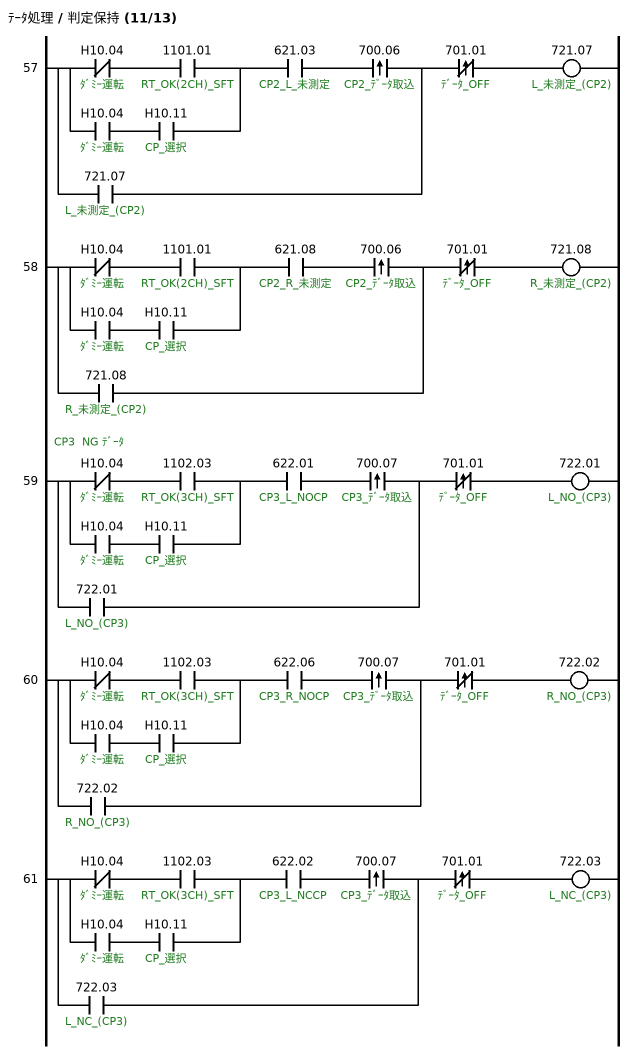
; [picture p144: ﾃｰﾀ処理 / 判定保持, rungs 57-61]
; rung 57
LDNOT H10.04  ; ﾀﾞﾐｰ運転
AND 1101.01  ; RT_OK(2CH)_SFT
LD H10.04  ; ﾀﾞﾐｰ運転
AND H10.11  ; CP_選択
ORLD
AND 621.03  ; CP2_L_未測定
@AND 700.06  ; CP2_ﾃﾞｰﾀ取込
OR 721.07  ; L_未測定_(CP2)
@ANDNOT 701.01  ; ﾃﾞｰﾀ_OFF
OUT 721.07  ; L_未測定_(CP2)
; rung 58
LDNOT H10.04  ; ﾀﾞﾐｰ運転
AND 1101.01  ; RT_OK(2CH)_SFT
LD H10.04  ; ﾀﾞﾐｰ運転
AND H10.11  ; CP_選択
ORLD
AND 621.08  ; CP2_R_未測定
@AND 700.06  ; CP2_ﾃﾞｰﾀ取込
OR 721.08  ; R_未測定_(CP2)
@ANDNOT 701.01  ; ﾃﾞｰﾀ_OFF
OUT 721.08  ; R_未測定_(CP2)
; rung 59: CP3  NG ﾃﾞｰﾀ
LDNOT H10.04  ; ﾀﾞﾐｰ運転
AND 1102.03  ; RT_OK(3CH)_SFT
LD H10.04  ; ﾀﾞﾐｰ運転
AND H10.11  ; CP_選択
ORLD
AND 622.01  ; CP3_L_NOCP
@AND 700.07  ; CP3_ﾃﾞｰﾀ取込
OR 722.01  ; L_NO_(CP3)
@ANDNOT 701.01  ; ﾃﾞｰﾀ_OFF
OUT 722.01  ; L_NO_(CP3)
; rung 60
LDNOT H10.04  ; ﾀﾞﾐｰ運転
AND 1102.03  ; RT_OK(3CH)_SFT
LD H10.04  ; ﾀﾞﾐｰ運転
AND H10.11  ; CP_選択
ORLD
AND 622.06  ; CP3_R_NOCP
@AND 700.07  ; CP3_ﾃﾞｰﾀ取込
OR 722.02  ; R_NO_(CP3)
@ANDNOT 701.01  ; ﾃﾞｰﾀ_OFF
OUT 722.02  ; R_NO_(CP3)
; rung 61
LDNOT H10.04  ; ﾀﾞﾐｰ運転
AND 1102.03  ; RT_OK(3CH)_SFT
LD H10.04  ; ﾀﾞﾐｰ運転
AND H10.11  ; CP_選択
ORLD
AND 622.02  ; CP3_L_NCCP
@AND 700.07  ; CP3_ﾃﾞｰﾀ取込
OR 722.03  ; L_NC_(CP3)
@ANDNOT 701.01  ; ﾃﾞｰﾀ_OFF
OUT 722.03  ; L_NC_(CP3)

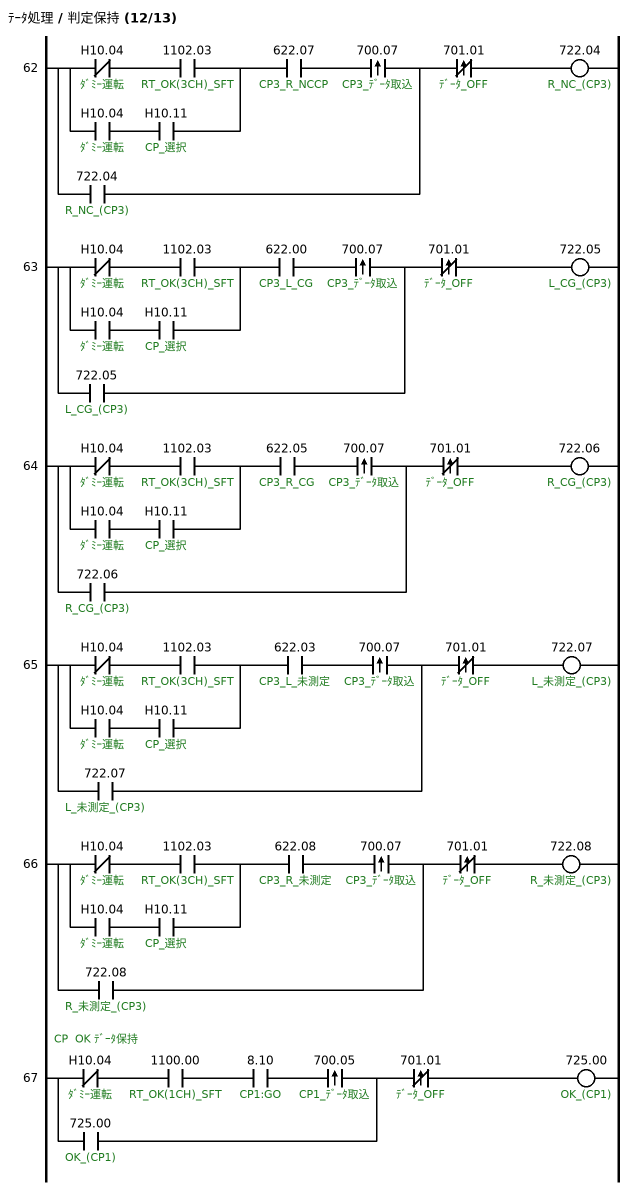
; rung 62
LDNOT H10.04  ; ﾀﾞﾐｰ運転
AND 1102.03  ; RT_OK(3CH)_SFT
LD H10.04  ; ﾀﾞﾐｰ運転
AND H10.11  ; CP_選択
ORLD
AND 622.07  ; CP3_R_NCCP
@AND 700.07  ; CP3_ﾃﾞｰﾀ取込
OR 722.04  ; R_NC_(CP3)
@ANDNOT 701.01  ; ﾃﾞｰﾀ_OFF
OUT 722.04  ; R_NC_(CP3)
; rung 63
LDNOT H10.04  ; ﾀﾞﾐｰ運転
AND 1102.03  ; RT_OK(3CH)_SFT
LD H10.04  ; ﾀﾞﾐｰ運転
AND H10.11  ; CP_選択
ORLD
AND 622.00  ; CP3_L_CG
@AND 700.07  ; CP3_ﾃﾞｰﾀ取込
OR 722.05  ; L_CG_(CP3)
@ANDNOT 701.01  ; ﾃﾞｰﾀ_OFF
OUT 722.05  ; L_CG_(CP3)
; rung 64
LDNOT H10.04  ; ﾀﾞﾐｰ運転
AND 1102.03  ; RT_OK(3CH)_SFT
LD H10.04  ; ﾀﾞﾐｰ運転
AND H10.11  ; CP_選択
ORLD
AND 622.05  ; CP3_R_CG
@AND 700.07  ; CP3_ﾃﾞｰﾀ取込
OR 722.06  ; R_CG_(CP3)
@ANDNOT 701.01  ; ﾃﾞｰﾀ_OFF
OUT 722.06  ; R_CG_(CP3)
; rung 65
LDNOT H10.04  ; ﾀﾞﾐｰ運転
AND 1102.03  ; RT_OK(3CH)_SFT
LD H10.04  ; ﾀﾞﾐｰ運転
AND H10.11  ; CP_選択
ORLD
AND 622.03  ; CP3_L_未測定
@AND 700.07  ; CP3_ﾃﾞｰﾀ取込
OR 722.07  ; L_未測定_(CP3)
@ANDNOT 701.01  ; ﾃﾞｰﾀ_OFF
OUT 722.07  ; L_未測定_(CP3)
; rung 66
LDNOT H10.04  ; ﾀﾞﾐｰ運転
AND 1102.03  ; RT_OK(3CH)_SFT
LD H10.04  ; ﾀﾞﾐｰ運転
AND H10.11  ; CP_選択
ORLD
AND 622.08  ; CP3_R_未測定
@AND 700.07  ; CP3_ﾃﾞｰﾀ取込
OR 722.08  ; R_未測定_(CP3)
@ANDNOT 701.01  ; ﾃﾞｰﾀ_OFF
OUT 722.08  ; R_未測定_(CP3)
; rung 67: CP  OK ﾃﾞｰﾀ保持
LDNOT H10.04  ; ﾀﾞﾐｰ運転
AND 1100.00  ; RT_OK(1CH)_SFT
AND 8.10  ; CP1:GO
@AND 700.05  ; CP1_ﾃﾞｰﾀ取込
OR 725.00  ; OK_(CP1)
@ANDNOT 701.01  ; ﾃﾞｰﾀ_OFF
OUT 725.00  ; OK_(CP1)

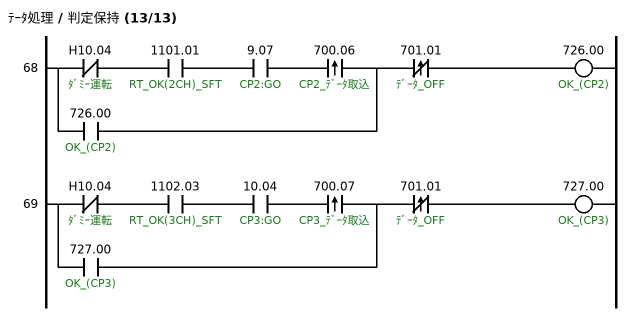
; rung 68
LDNOT H10.04  ; ﾀﾞﾐｰ運転
AND 1101.01  ; RT_OK(2CH)_SFT
AND 9.07  ; CP2:GO
@AND 700.06  ; CP2_ﾃﾞｰﾀ取込
OR 726.00  ; OK_(CP2)
@ANDNOT 701.01  ; ﾃﾞｰﾀ_OFF
OUT 726.00  ; OK_(CP2)
; rung 69
LDNOT H10.04  ; ﾀﾞﾐｰ運転
AND 1102.03  ; RT_OK(3CH)_SFT
AND 10.04  ; CP3:GO
@AND 700.07  ; CP3_ﾃﾞｰﾀ取込
OR 727.00  ; OK_(CP3)
@ANDNOT 701.01  ; ﾃﾞｰﾀ_OFF
OUT 727.00  ; OK_(CP3)

### Section NG_SFT

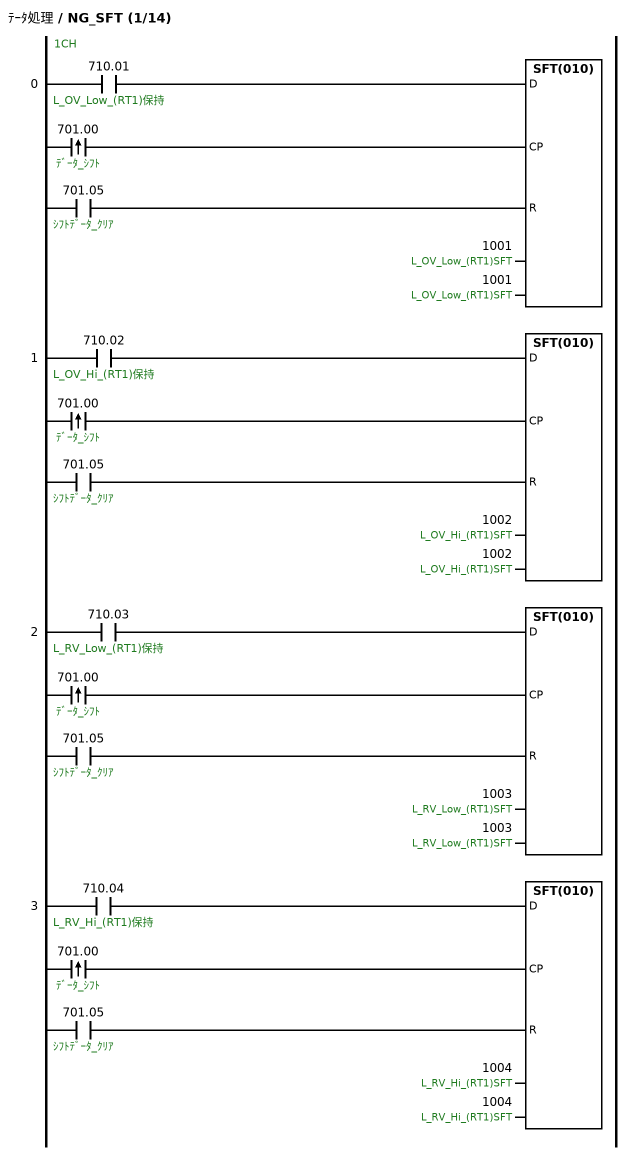
; rung 0: 1CH
LD 710.01  ; L_OV_Low_(RT1)保持
@LD 701.00  ; ﾃﾞｰﾀ_ｼﾌﾄ
LD 701.05  ; ｼﾌﾄﾃﾞｰﾀ_ｸﾘｱ
SFT(010) 1001 1001  ; L_OV_Low_(RT1)SFT
; rung 1
LD 710.02  ; L_OV_Hi_(RT1)保持
@LD 701.00  ; ﾃﾞｰﾀ_ｼﾌﾄ
LD 701.05  ; ｼﾌﾄﾃﾞｰﾀ_ｸﾘｱ
SFT(010) 1002 1002  ; L_OV_Hi_(RT1)SFT
; rung 2
LD 710.03  ; L_RV_Low_(RT1)保持
@LD 701.00  ; ﾃﾞｰﾀ_ｼﾌﾄ
LD 701.05  ; ｼﾌﾄﾃﾞｰﾀ_ｸﾘｱ
SFT(010) 1003 1003  ; L_RV_Low_(RT1)SFT
; rung 3
LD 710.04  ; L_RV_Hi_(RT1)保持
@LD 701.00  ; ﾃﾞｰﾀ_ｼﾌﾄ
LD 701.05  ; ｼﾌﾄﾃﾞｰﾀ_ｸﾘｱ
SFT(010) 1004 1004  ; L_RV_Hi_(RT1)SFT

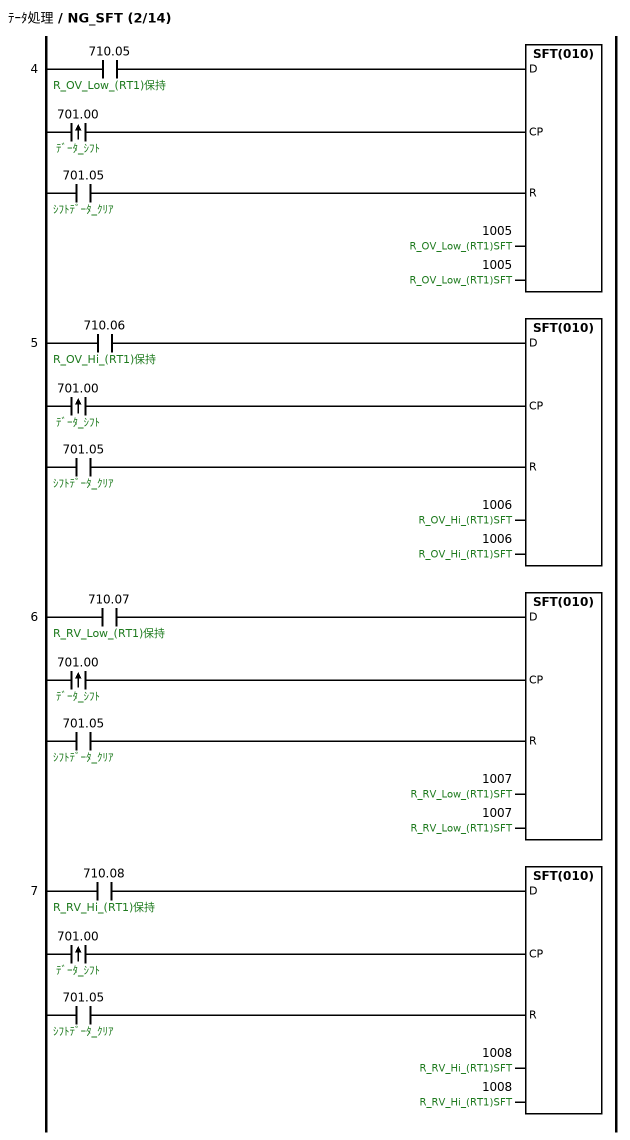
; rung 4
LD 710.05  ; R_OV_Low_(RT1)保持
@LD 701.00  ; ﾃﾞｰﾀ_ｼﾌﾄ
LD 701.05  ; ｼﾌﾄﾃﾞｰﾀ_ｸﾘｱ
SFT(010) 1005 1005  ; R_OV_Low_(RT1)SFT
; rung 5
LD 710.06  ; R_OV_Hi_(RT1)保持
@LD 701.00  ; ﾃﾞｰﾀ_ｼﾌﾄ
LD 701.05  ; ｼﾌﾄﾃﾞｰﾀ_ｸﾘｱ
SFT(010) 1006 1006  ; R_OV_Hi_(RT1)SFT
; rung 6
LD 710.07  ; R_RV_Low_(RT1)保持
@LD 701.00  ; ﾃﾞｰﾀ_ｼﾌﾄ
LD 701.05  ; ｼﾌﾄﾃﾞｰﾀ_ｸﾘｱ
SFT(010) 1007 1007  ; R_RV_Low_(RT1)SFT
; rung 7
LD 710.08  ; R_RV_Hi_(RT1)保持
@LD 701.00  ; ﾃﾞｰﾀ_ｼﾌﾄ
LD 701.05  ; ｼﾌﾄﾃﾞｰﾀ_ｸﾘｱ
SFT(010) 1008 1008  ; R_RV_Hi_(RT1)SFT

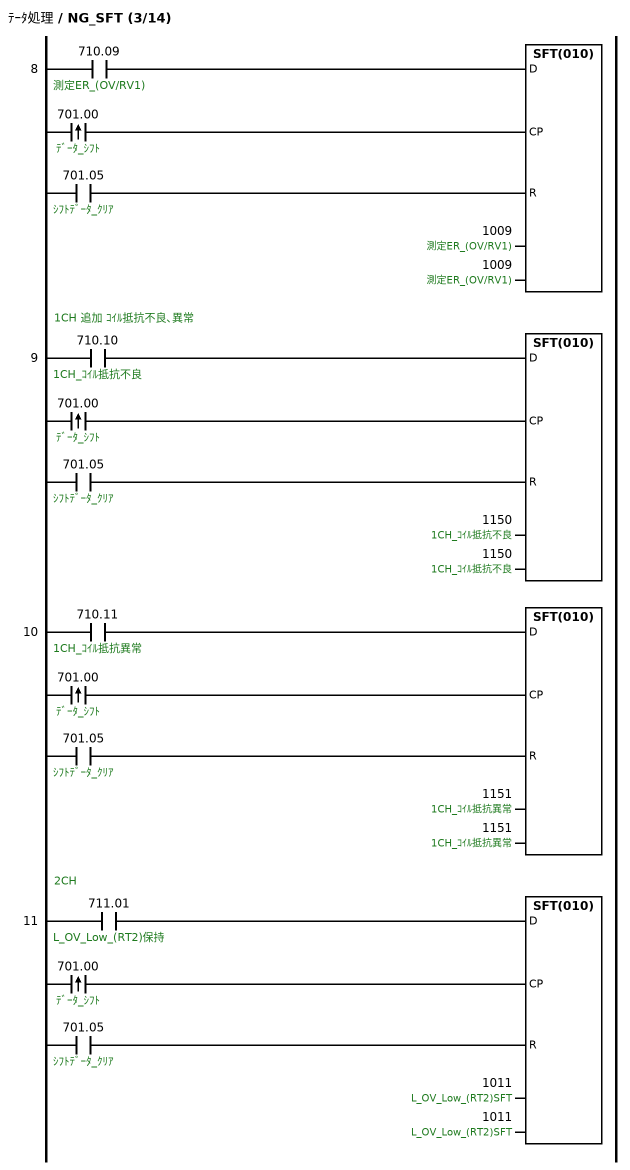
; rung 8
LD 710.09  ; 測定ER_(OV/RV1)
@LD 701.00  ; ﾃﾞｰﾀ_ｼﾌﾄ
LD 701.05  ; ｼﾌﾄﾃﾞｰﾀ_ｸﾘｱ
SFT(010) 1009 1009  ; 測定ER_(OV/RV1)
; rung 9: 1CH 追加 ｺｲﾙ抵抗不良､異常
LD 710.10  ; 1CH_ｺｲﾙ抵抗不良
@LD 701.00  ; ﾃﾞｰﾀ_ｼﾌﾄ
LD 701.05  ; ｼﾌﾄﾃﾞｰﾀ_ｸﾘｱ
SFT(010) 1150 1150  ; 1CH_ｺｲﾙ抵抗不良
; rung 10
LD 710.11  ; 1CH_ｺｲﾙ抵抗異常
@LD 701.00  ; ﾃﾞｰﾀ_ｼﾌﾄ
LD 701.05  ; ｼﾌﾄﾃﾞｰﾀ_ｸﾘｱ
SFT(010) 1151 1151  ; 1CH_ｺｲﾙ抵抗異常
; rung 11: 2CH
LD 711.01  ; L_OV_Low_(RT2)保持
@LD 701.00  ; ﾃﾞｰﾀ_ｼﾌﾄ
LD 701.05  ; ｼﾌﾄﾃﾞｰﾀ_ｸﾘｱ
SFT(010) 1011 1011  ; L_OV_Low_(RT2)SFT

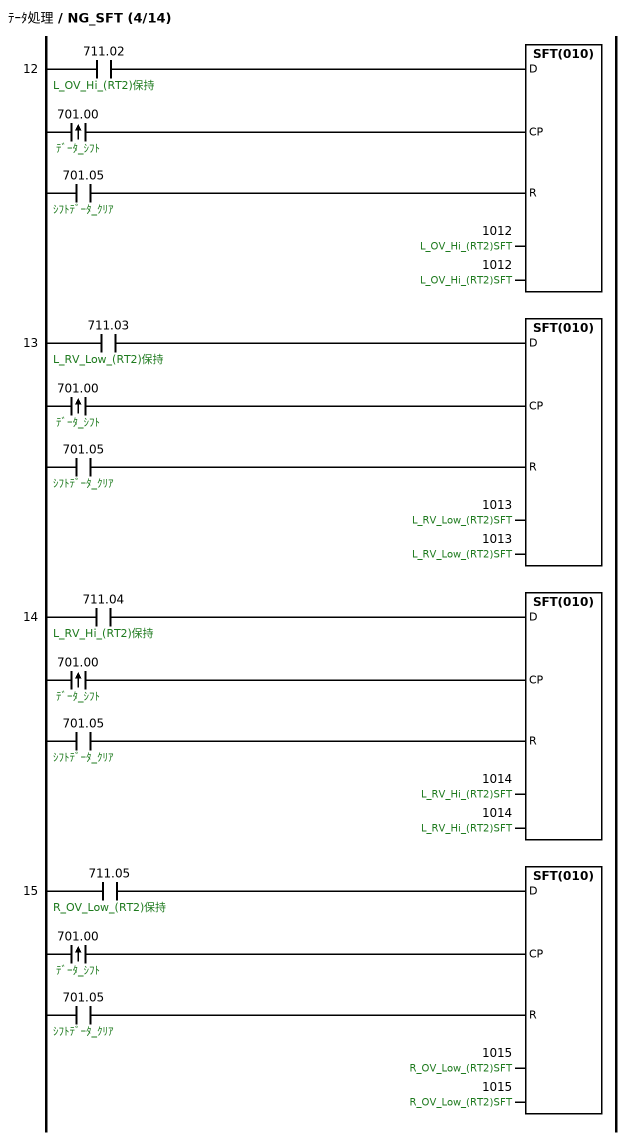
; rung 12
LD 711.02  ; L_OV_Hi_(RT2)保持
@LD 701.00  ; ﾃﾞｰﾀ_ｼﾌﾄ
LD 701.05  ; ｼﾌﾄﾃﾞｰﾀ_ｸﾘｱ
SFT(010) 1012 1012  ; L_OV_Hi_(RT2)SFT
; rung 13
LD 711.03  ; L_RV_Low_(RT2)保持
@LD 701.00  ; ﾃﾞｰﾀ_ｼﾌﾄ
LD 701.05  ; ｼﾌﾄﾃﾞｰﾀ_ｸﾘｱ
SFT(010) 1013 1013  ; L_RV_Low_(RT2)SFT
; rung 14
LD 711.04  ; L_RV_Hi_(RT2)保持
@LD 701.00  ; ﾃﾞｰﾀ_ｼﾌﾄ
LD 701.05  ; ｼﾌﾄﾃﾞｰﾀ_ｸﾘｱ
SFT(010) 1014 1014  ; L_RV_Hi_(RT2)SFT
; rung 15
LD 711.05  ; R_OV_Low_(RT2)保持
@LD 701.00  ; ﾃﾞｰﾀ_ｼﾌﾄ
LD 701.05  ; ｼﾌﾄﾃﾞｰﾀ_ｸﾘｱ
SFT(010) 1015 1015  ; R_OV_Low_(RT2)SFT

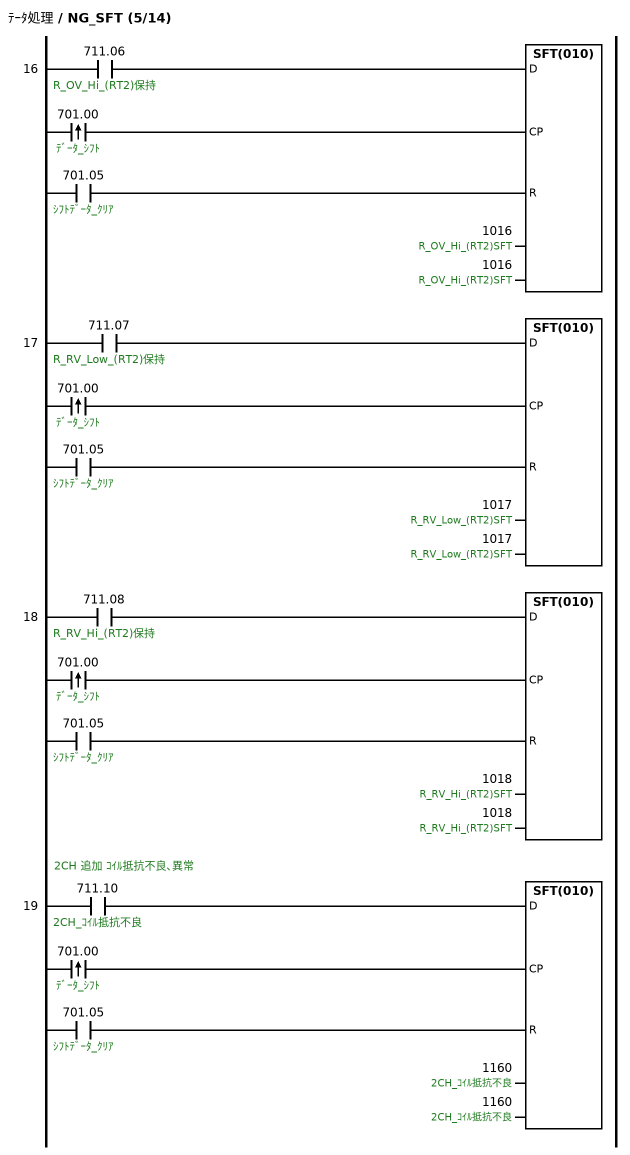
; rung 16
LD 711.06  ; R_OV_Hi_(RT2)保持
@LD 701.00  ; ﾃﾞｰﾀ_ｼﾌﾄ
LD 701.05  ; ｼﾌﾄﾃﾞｰﾀ_ｸﾘｱ
SFT(010) 1016 1016  ; R_OV_Hi_(RT2)SFT
; rung 17
LD 711.07  ; R_RV_Low_(RT2)保持
@LD 701.00  ; ﾃﾞｰﾀ_ｼﾌﾄ
LD 701.05  ; ｼﾌﾄﾃﾞｰﾀ_ｸﾘｱ
SFT(010) 1017 1017  ; R_RV_Low_(RT2)SFT
; rung 18
LD 711.08  ; R_RV_Hi_(RT2)保持
@LD 701.00  ; ﾃﾞｰﾀ_ｼﾌﾄ
LD 701.05  ; ｼﾌﾄﾃﾞｰﾀ_ｸﾘｱ
SFT(010) 1018 1018  ; R_RV_Hi_(RT2)SFT
; rung 19: 2CH 追加 ｺｲﾙ抵抗不良､異常
LD 711.10  ; 2CH_ｺｲﾙ抵抗不良
@LD 701.00  ; ﾃﾞｰﾀ_ｼﾌﾄ
LD 701.05  ; ｼﾌﾄﾃﾞｰﾀ_ｸﾘｱ
SFT(010) 1160 1160  ; 2CH_ｺｲﾙ抵抗不良

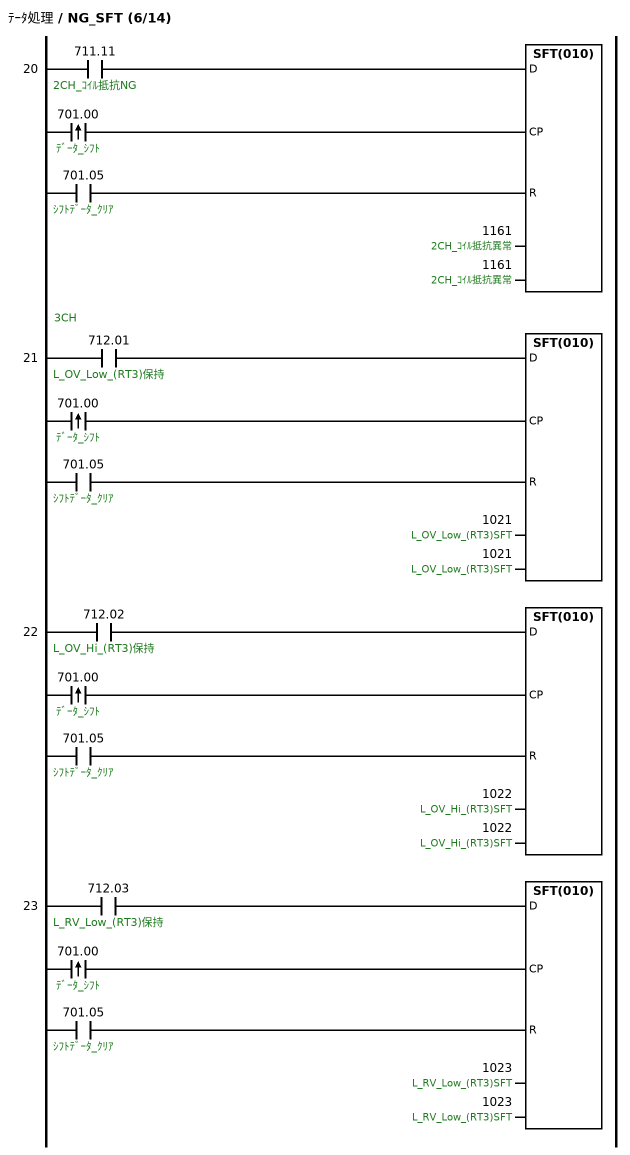
; rung 20
LD 711.11  ; 2CH_ｺｲﾙ抵抗NG
@LD 701.00  ; ﾃﾞｰﾀ_ｼﾌﾄ
LD 701.05  ; ｼﾌﾄﾃﾞｰﾀ_ｸﾘｱ
SFT(010) 1161 1161  ; 2CH_ｺｲﾙ抵抗異常
; rung 21: 3CH
LD 712.01  ; L_OV_Low_(RT3)保持
@LD 701.00  ; ﾃﾞｰﾀ_ｼﾌﾄ
LD 701.05  ; ｼﾌﾄﾃﾞｰﾀ_ｸﾘｱ
SFT(010) 1021 1021  ; L_OV_Low_(RT3)SFT
; rung 22
LD 712.02  ; L_OV_Hi_(RT3)保持
@LD 701.00  ; ﾃﾞｰﾀ_ｼﾌﾄ
LD 701.05  ; ｼﾌﾄﾃﾞｰﾀ_ｸﾘｱ
SFT(010) 1022 1022  ; L_OV_Hi_(RT3)SFT
; rung 23
LD 712.03  ; L_RV_Low_(RT3)保持
@LD 701.00  ; ﾃﾞｰﾀ_ｼﾌﾄ
LD 701.05  ; ｼﾌﾄﾃﾞｰﾀ_ｸﾘｱ
SFT(010) 1023 1023  ; L_RV_Low_(RT3)SFT

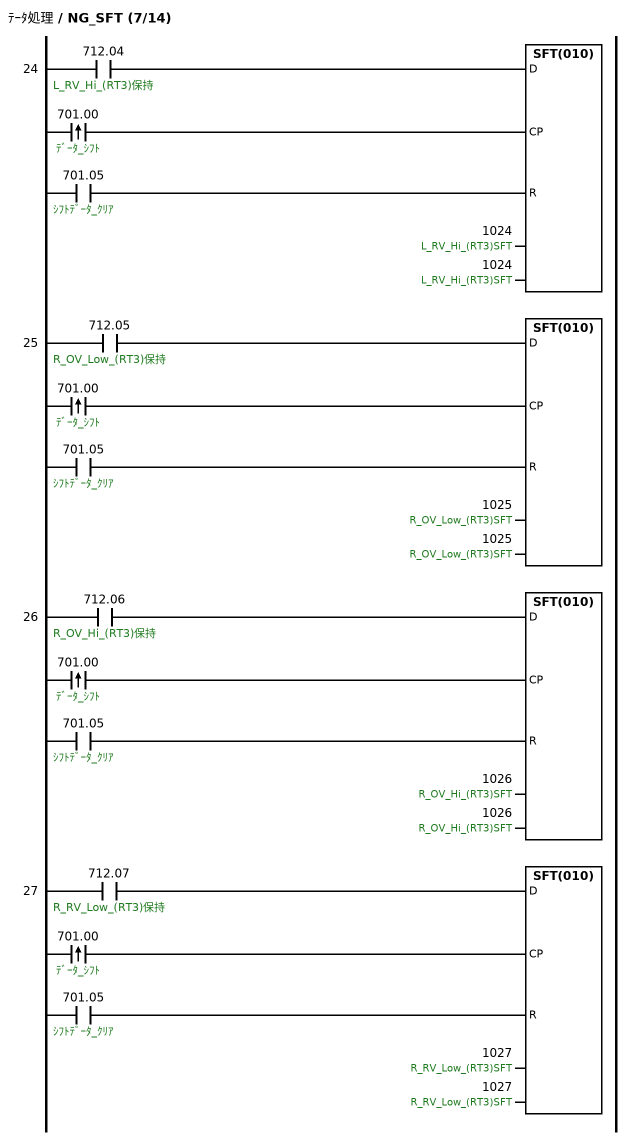
; rung 24
LD 712.04  ; L_RV_Hi_(RT3)保持
@LD 701.00  ; ﾃﾞｰﾀ_ｼﾌﾄ
LD 701.05  ; ｼﾌﾄﾃﾞｰﾀ_ｸﾘｱ
SFT(010) 1024 1024  ; L_RV_Hi_(RT3)SFT
; rung 25
LD 712.05  ; R_OV_Low_(RT3)保持
@LD 701.00  ; ﾃﾞｰﾀ_ｼﾌﾄ
LD 701.05  ; ｼﾌﾄﾃﾞｰﾀ_ｸﾘｱ
SFT(010) 1025 1025  ; R_OV_Low_(RT3)SFT
; rung 26
LD 712.06  ; R_OV_Hi_(RT3)保持
@LD 701.00  ; ﾃﾞｰﾀ_ｼﾌﾄ
LD 701.05  ; ｼﾌﾄﾃﾞｰﾀ_ｸﾘｱ
SFT(010) 1026 1026  ; R_OV_Hi_(RT3)SFT
; rung 27
LD 712.07  ; R_RV_Low_(RT3)保持
@LD 701.00  ; ﾃﾞｰﾀ_ｼﾌﾄ
LD 701.05  ; ｼﾌﾄﾃﾞｰﾀ_ｸﾘｱ
SFT(010) 1027 1027  ; R_RV_Low_(RT3)SFT

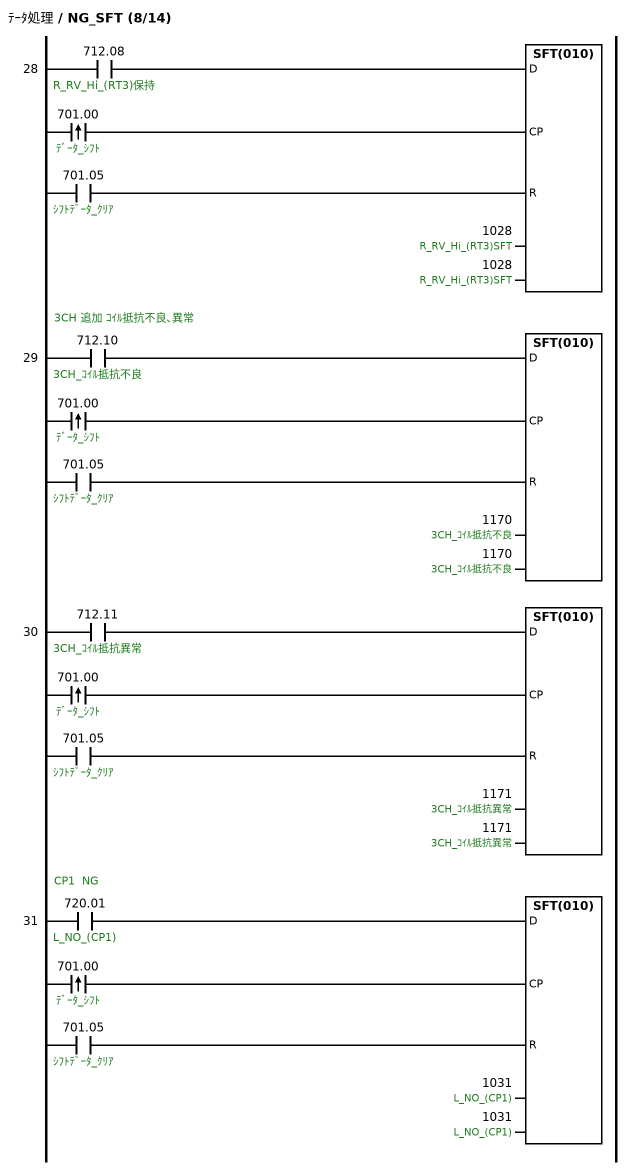
; rung 28
LD 712.08  ; R_RV_Hi_(RT3)保持
@LD 701.00  ; ﾃﾞｰﾀ_ｼﾌﾄ
LD 701.05  ; ｼﾌﾄﾃﾞｰﾀ_ｸﾘｱ
SFT(010) 1028 1028  ; R_RV_Hi_(RT3)SFT
; rung 29: 3CH 追加 ｺｲﾙ抵抗不良､異常
LD 712.10  ; 3CH_ｺｲﾙ抵抗不良
@LD 701.00  ; ﾃﾞｰﾀ_ｼﾌﾄ
LD 701.05  ; ｼﾌﾄﾃﾞｰﾀ_ｸﾘｱ
SFT(010) 1170 1170  ; 3CH_ｺｲﾙ抵抗不良
; rung 30
LD 712.11  ; 3CH_ｺｲﾙ抵抗異常
@LD 701.00  ; ﾃﾞｰﾀ_ｼﾌﾄ
LD 701.05  ; ｼﾌﾄﾃﾞｰﾀ_ｸﾘｱ
SFT(010) 1171 1171  ; 3CH_ｺｲﾙ抵抗異常
; rung 31: CP1  NG
LD 720.01  ; L_NO_(CP1)
@LD 701.00  ; ﾃﾞｰﾀ_ｼﾌﾄ
LD 701.05  ; ｼﾌﾄﾃﾞｰﾀ_ｸﾘｱ
SFT(010) 1031 1031  ; L_NO_(CP1)

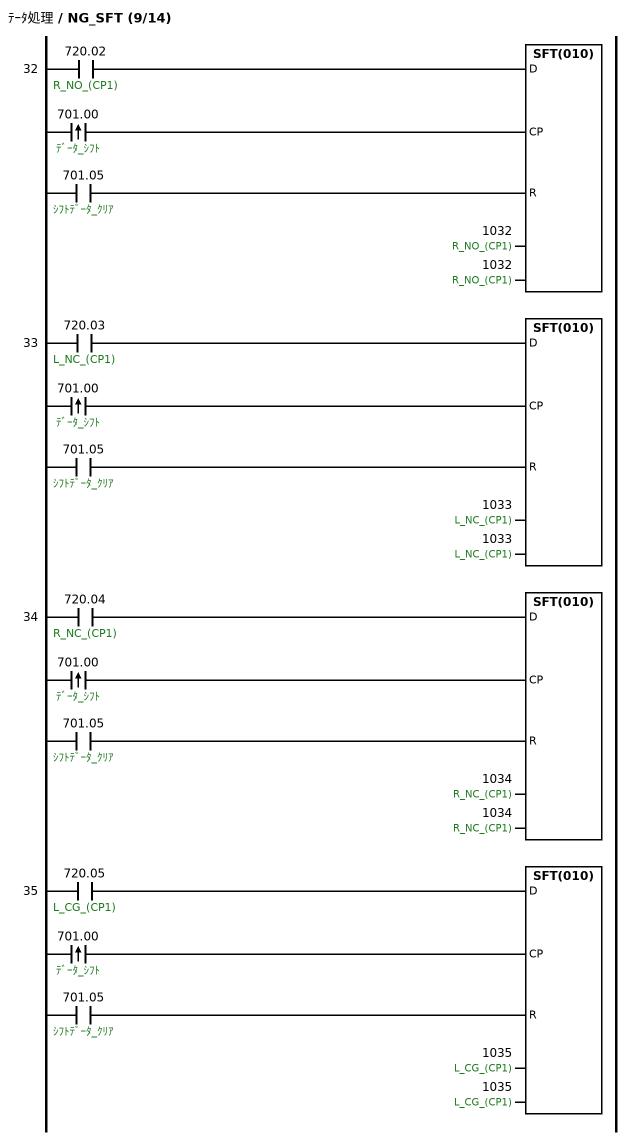
; rung 32
LD 720.02  ; R_NO_(CP1)
@LD 701.00  ; ﾃﾞｰﾀ_ｼﾌﾄ
LD 701.05  ; ｼﾌﾄﾃﾞｰﾀ_ｸﾘｱ
SFT(010) 1032 1032  ; R_NO_(CP1)
; rung 33
LD 720.03  ; L_NC_(CP1)
@LD 701.00  ; ﾃﾞｰﾀ_ｼﾌﾄ
LD 701.05  ; ｼﾌﾄﾃﾞｰﾀ_ｸﾘｱ
SFT(010) 1033 1033  ; L_NC_(CP1)
; rung 34
LD 720.04  ; R_NC_(CP1)
@LD 701.00  ; ﾃﾞｰﾀ_ｼﾌﾄ
LD 701.05  ; ｼﾌﾄﾃﾞｰﾀ_ｸﾘｱ
SFT(010) 1034 1034  ; R_NC_(CP1)
; rung 35
LD 720.05  ; L_CG_(CP1)
@LD 701.00  ; ﾃﾞｰﾀ_ｼﾌﾄ
LD 701.05  ; ｼﾌﾄﾃﾞｰﾀ_ｸﾘｱ
SFT(010) 1035 1035  ; L_CG_(CP1)

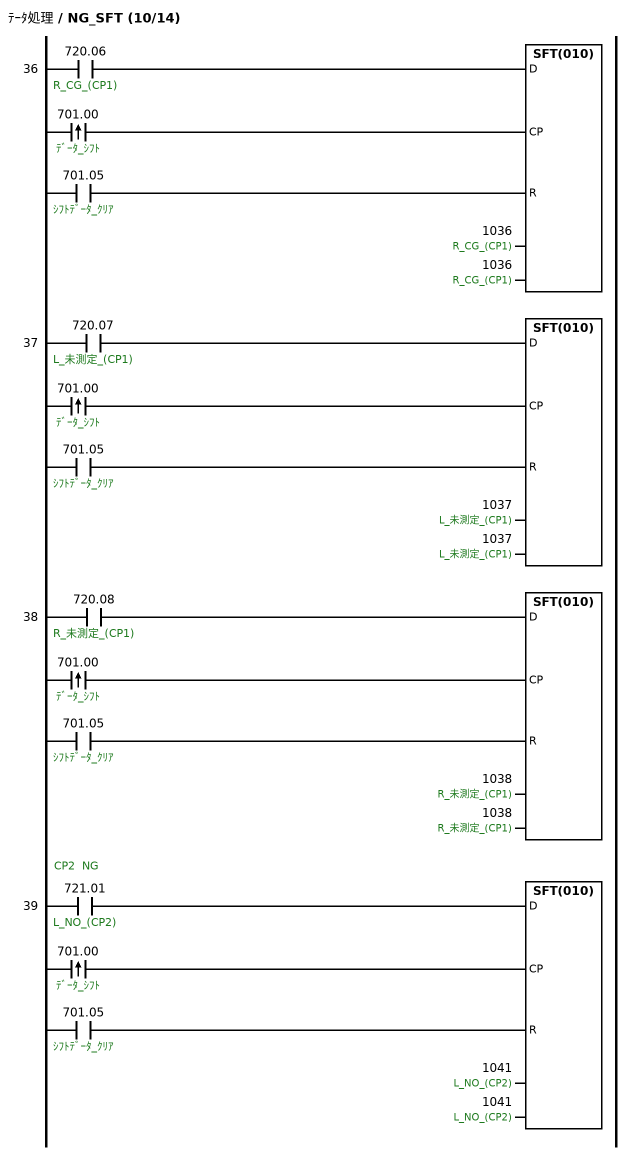
; rung 36
LD 720.06  ; R_CG_(CP1)
@LD 701.00  ; ﾃﾞｰﾀ_ｼﾌﾄ
LD 701.05  ; ｼﾌﾄﾃﾞｰﾀ_ｸﾘｱ
SFT(010) 1036 1036  ; R_CG_(CP1)
; rung 37
LD 720.07  ; L_未測定_(CP1)
@LD 701.00  ; ﾃﾞｰﾀ_ｼﾌﾄ
LD 701.05  ; ｼﾌﾄﾃﾞｰﾀ_ｸﾘｱ
SFT(010) 1037 1037  ; L_未測定_(CP1)
; rung 38
LD 720.08  ; R_未測定_(CP1)
@LD 701.00  ; ﾃﾞｰﾀ_ｼﾌﾄ
LD 701.05  ; ｼﾌﾄﾃﾞｰﾀ_ｸﾘｱ
SFT(010) 1038 1038  ; R_未測定_(CP1)
; rung 39: CP2  NG
LD 721.01  ; L_NO_(CP2)
@LD 701.00  ; ﾃﾞｰﾀ_ｼﾌﾄ
LD 701.05  ; ｼﾌﾄﾃﾞｰﾀ_ｸﾘｱ
SFT(010) 1041 1041  ; L_NO_(CP2)

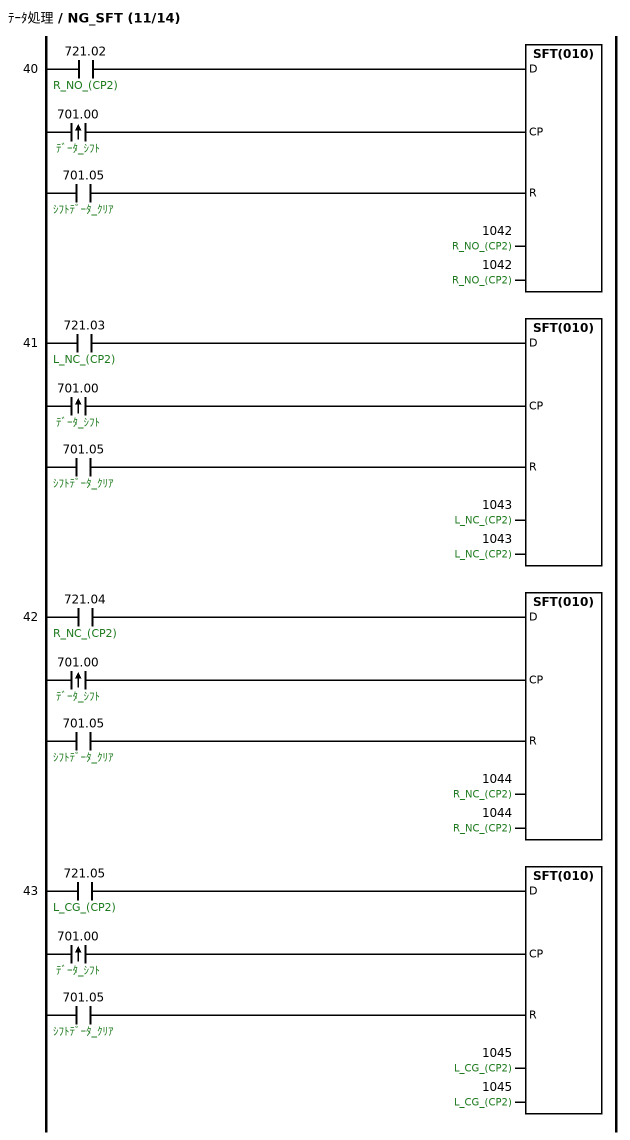
; rung 40
LD 721.02  ; R_NO_(CP2)
@LD 701.00  ; ﾃﾞｰﾀ_ｼﾌﾄ
LD 701.05  ; ｼﾌﾄﾃﾞｰﾀ_ｸﾘｱ
SFT(010) 1042 1042  ; R_NO_(CP2)
; rung 41
LD 721.03  ; L_NC_(CP2)
@LD 701.00  ; ﾃﾞｰﾀ_ｼﾌﾄ
LD 701.05  ; ｼﾌﾄﾃﾞｰﾀ_ｸﾘｱ
SFT(010) 1043 1043  ; L_NC_(CP2)
; rung 42
LD 721.04  ; R_NC_(CP2)
@LD 701.00  ; ﾃﾞｰﾀ_ｼﾌﾄ
LD 701.05  ; ｼﾌﾄﾃﾞｰﾀ_ｸﾘｱ
SFT(010) 1044 1044  ; R_NC_(CP2)
; rung 43
LD 721.05  ; L_CG_(CP2)
@LD 701.00  ; ﾃﾞｰﾀ_ｼﾌﾄ
LD 701.05  ; ｼﾌﾄﾃﾞｰﾀ_ｸﾘｱ
SFT(010) 1045 1045  ; L_CG_(CP2)

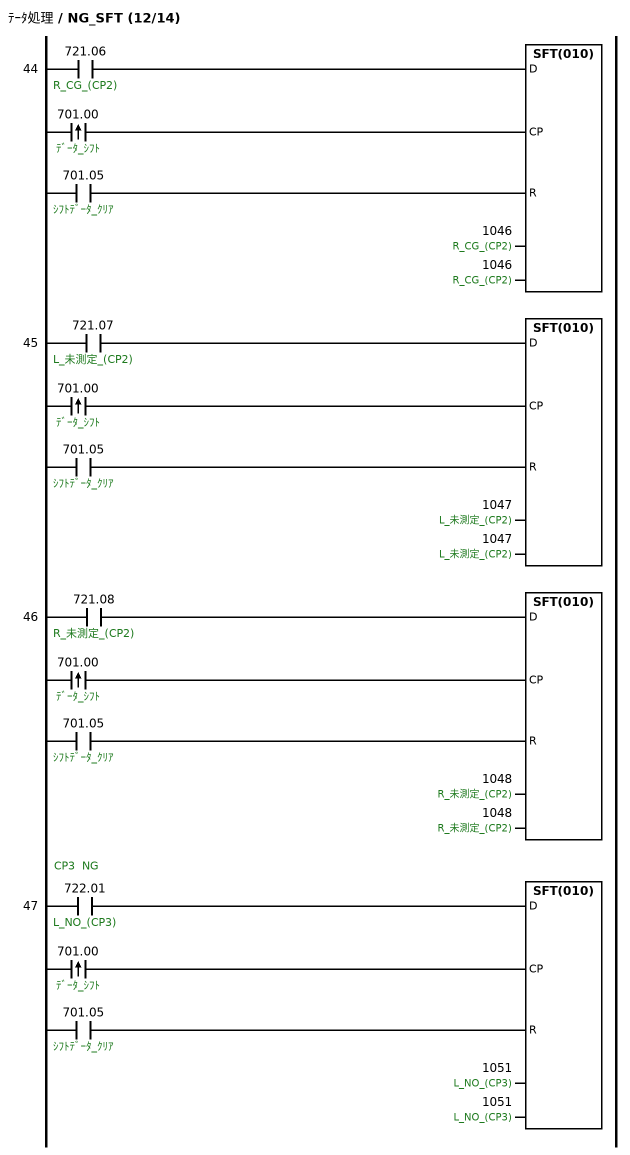
; rung 44
LD 721.06  ; R_CG_(CP2)
@LD 701.00  ; ﾃﾞｰﾀ_ｼﾌﾄ
LD 701.05  ; ｼﾌﾄﾃﾞｰﾀ_ｸﾘｱ
SFT(010) 1046 1046  ; R_CG_(CP2)
; rung 45
LD 721.07  ; L_未測定_(CP2)
@LD 701.00  ; ﾃﾞｰﾀ_ｼﾌﾄ
LD 701.05  ; ｼﾌﾄﾃﾞｰﾀ_ｸﾘｱ
SFT(010) 1047 1047  ; L_未測定_(CP2)
; rung 46
LD 721.08  ; R_未測定_(CP2)
@LD 701.00  ; ﾃﾞｰﾀ_ｼﾌﾄ
LD 701.05  ; ｼﾌﾄﾃﾞｰﾀ_ｸﾘｱ
SFT(010) 1048 1048  ; R_未測定_(CP2)
; rung 47: CP3  NG
LD 722.01  ; L_NO_(CP3)
@LD 701.00  ; ﾃﾞｰﾀ_ｼﾌﾄ
LD 701.05  ; ｼﾌﾄﾃﾞｰﾀ_ｸﾘｱ
SFT(010) 1051 1051  ; L_NO_(CP3)

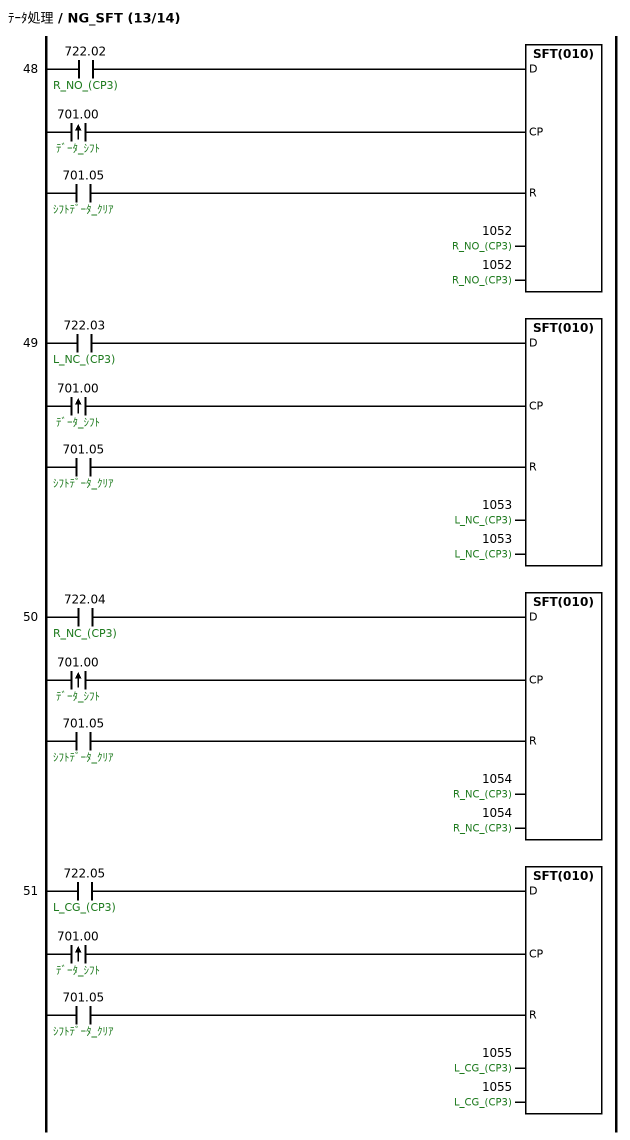
; rung 48
LD 722.02  ; R_NO_(CP3)
@LD 701.00  ; ﾃﾞｰﾀ_ｼﾌﾄ
LD 701.05  ; ｼﾌﾄﾃﾞｰﾀ_ｸﾘｱ
SFT(010) 1052 1052  ; R_NO_(CP3)
; rung 49
LD 722.03  ; L_NC_(CP3)
@LD 701.00  ; ﾃﾞｰﾀ_ｼﾌﾄ
LD 701.05  ; ｼﾌﾄﾃﾞｰﾀ_ｸﾘｱ
SFT(010) 1053 1053  ; L_NC_(CP3)
; rung 50
LD 722.04  ; R_NC_(CP3)
@LD 701.00  ; ﾃﾞｰﾀ_ｼﾌﾄ
LD 701.05  ; ｼﾌﾄﾃﾞｰﾀ_ｸﾘｱ
SFT(010) 1054 1054  ; R_NC_(CP3)
; rung 51
LD 722.05  ; L_CG_(CP3)
@LD 701.00  ; ﾃﾞｰﾀ_ｼﾌﾄ
LD 701.05  ; ｼﾌﾄﾃﾞｰﾀ_ｸﾘｱ
SFT(010) 1055 1055  ; L_CG_(CP3)

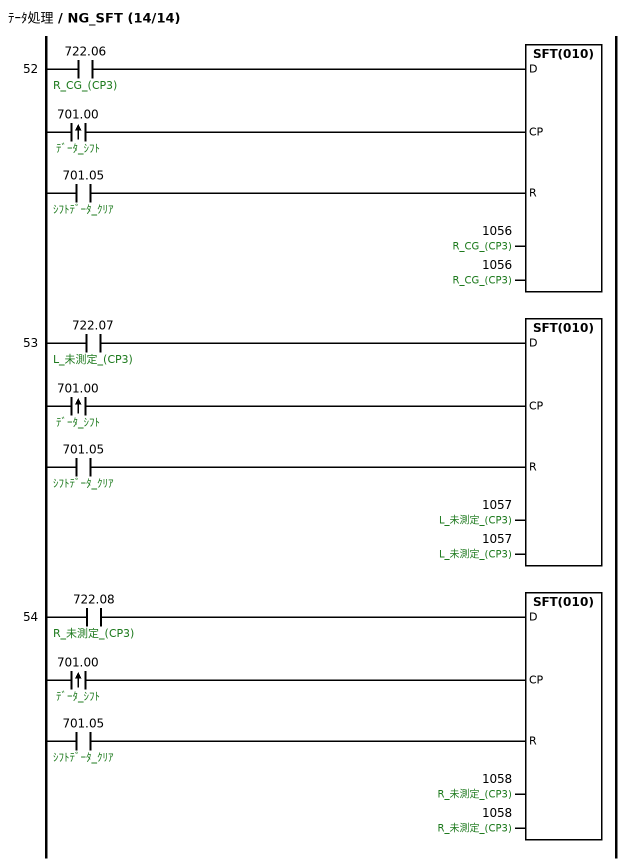
; rung 52
LD 722.06  ; R_CG_(CP3)
@LD 701.00  ; ﾃﾞｰﾀ_ｼﾌﾄ
LD 701.05  ; ｼﾌﾄﾃﾞｰﾀ_ｸﾘｱ
SFT(010) 1056 1056  ; R_CG_(CP3)
; rung 53
LD 722.07  ; L_未測定_(CP3)
@LD 701.00  ; ﾃﾞｰﾀ_ｼﾌﾄ
LD 701.05  ; ｼﾌﾄﾃﾞｰﾀ_ｸﾘｱ
SFT(010) 1057 1057  ; L_未測定_(CP3)
; rung 54
LD 722.08  ; R_未測定_(CP3)
@LD 701.00  ; ﾃﾞｰﾀ_ｼﾌﾄ
LD 701.05  ; ｼﾌﾄﾃﾞｰﾀ_ｸﾘｱ
SFT(010) 1058 1058  ; R_未測定_(CP3)

### Section OK_SFT

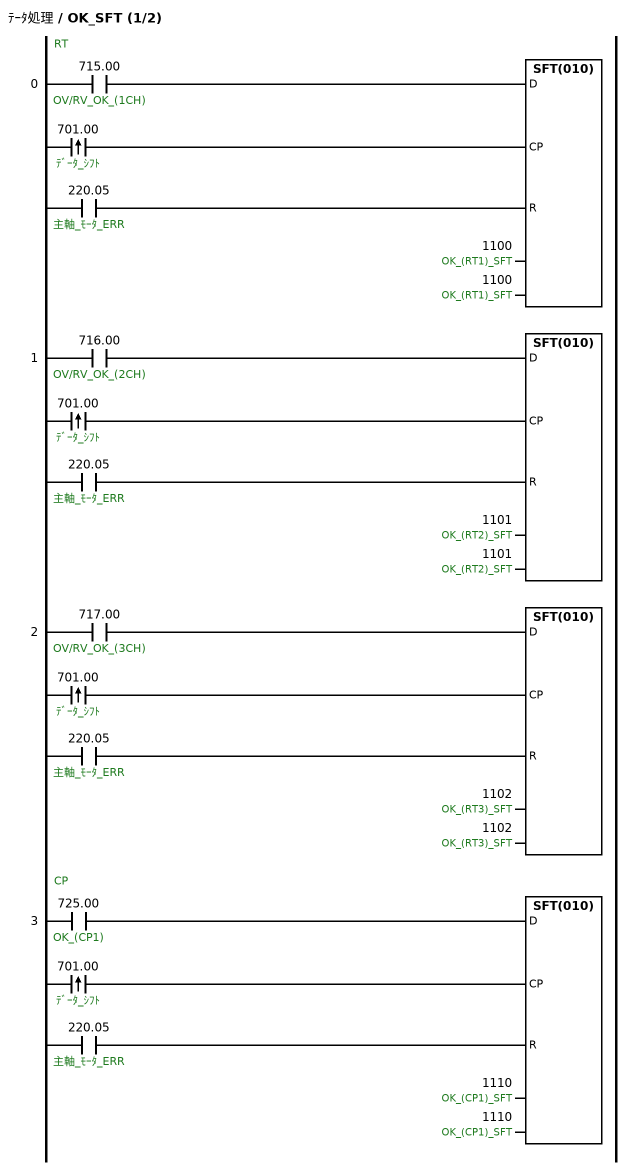
; rung 0: RT
LD 715.00  ; OV/RV_OK_(1CH)
@LD 701.00  ; ﾃﾞｰﾀ_ｼﾌﾄ
LD 220.05  ; 主軸_ﾓｰﾀ_ERR
SFT(010) 1100 1100  ; OK_(RT1)_SFT
; rung 1
LD 716.00  ; OV/RV_OK_(2CH)
@LD 701.00  ; ﾃﾞｰﾀ_ｼﾌﾄ
LD 220.05  ; 主軸_ﾓｰﾀ_ERR
SFT(010) 1101 1101  ; OK_(RT2)_SFT
; rung 2
LD 717.00  ; OV/RV_OK_(3CH)
@LD 701.00  ; ﾃﾞｰﾀ_ｼﾌﾄ
LD 220.05  ; 主軸_ﾓｰﾀ_ERR
SFT(010) 1102 1102  ; OK_(RT3)_SFT
; rung 3: CP
LD 725.00  ; OK_(CP1)
@LD 701.00  ; ﾃﾞｰﾀ_ｼﾌﾄ
LD 220.05  ; 主軸_ﾓｰﾀ_ERR
SFT(010) 1110 1110  ; OK_(CP1)_SFT

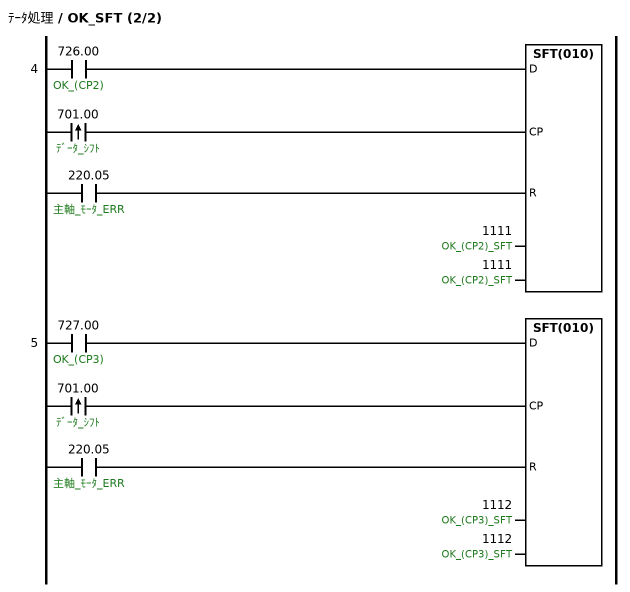
; rung 4
LD 726.00  ; OK_(CP2)
@LD 701.00  ; ﾃﾞｰﾀ_ｼﾌﾄ
LD 220.05  ; 主軸_ﾓｰﾀ_ERR
SFT(010) 1111 1111  ; OK_(CP2)_SFT
; rung 5
LD 727.00  ; OK_(CP3)
@LD 701.00  ; ﾃﾞｰﾀ_ｼﾌﾄ
LD 220.05  ; 主軸_ﾓｰﾀ_ERR
SFT(010) 1112 1112  ; OK_(CP3)_SFT

### Section ﾃﾞｰﾀ処理

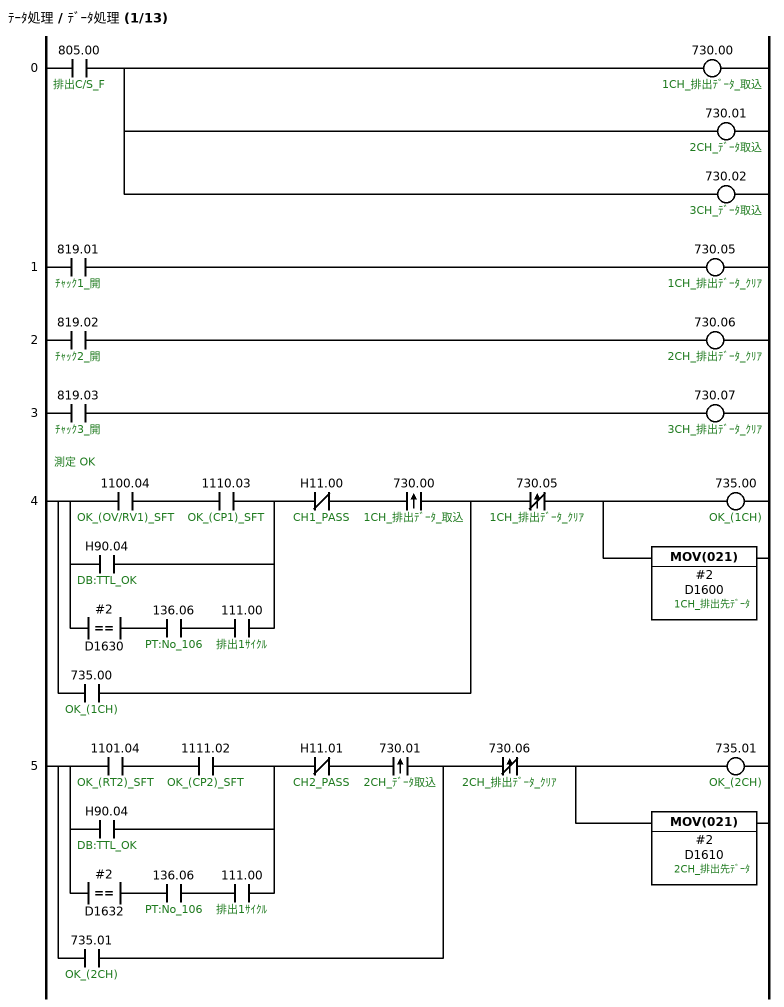
; rung 0
LD 805.00  ; 排出C/S_F
OUT 730.00  ; 1CH_排出ﾃﾞｰﾀ_取込
OUT 730.01  ; 2CH_ﾃﾞｰﾀ取込
OUT 730.02  ; 3CH_ﾃﾞｰﾀ取込
; rung 1
LD 819.01  ; ﾁｬｯｸ1_開
OUT 730.05  ; 1CH_排出ﾃﾞｰﾀ_ｸﾘｱ
; rung 2
LD 819.02  ; ﾁｬｯｸ2_開
OUT 730.06  ; 2CH_排出ﾃﾞｰﾀ_ｸﾘｱ
; rung 3
LD 819.03  ; ﾁｬｯｸ3_開
OUT 730.07  ; 3CH_排出ﾃﾞｰﾀ_ｸﾘｱ
; rung 4: 測定 OK
LD 1100.04  ; OK_(OV/RV1)_SFT
AND 1110.03  ; OK_(CP1)_SFT
OR H90.04  ; DB:TTL_OK
LD=(300) #2 D1630
AND 136.06  ; PT:No_106
AND 111.00  ; 排出1ｻｲｸﾙ
ORLD
ANDNOT H11.00  ; CH1_PASS
@AND 730.00  ; 1CH_排出ﾃﾞｰﾀ_取込
OR 735.00  ; OK_(1CH)
@ANDNOT 730.05  ; 1CH_排出ﾃﾞｰﾀ_ｸﾘｱ
OUT 735.00  ; OK_(1CH)
MOV(021) #2 D1600  ; 1CH_排出先ﾃﾞｰﾀ
; rung 5
LD 1101.04  ; OK_(RT2)_SFT
AND 1111.02  ; OK_(CP2)_SFT
OR H90.04  ; DB:TTL_OK
LD=(300) #2 D1632
AND 136.06  ; PT:No_106
AND 111.00  ; 排出1ｻｲｸﾙ
ORLD
ANDNOT H11.01  ; CH2_PASS
@AND 730.01  ; 2CH_ﾃﾞｰﾀ取込
OR 735.01  ; OK_(2CH)
@ANDNOT 730.06  ; 2CH_排出ﾃﾞｰﾀ_ｸﾘｱ
OUT 735.01  ; OK_(2CH)
MOV(021) #2 D1610  ; 2CH_排出先ﾃﾞｰﾀ

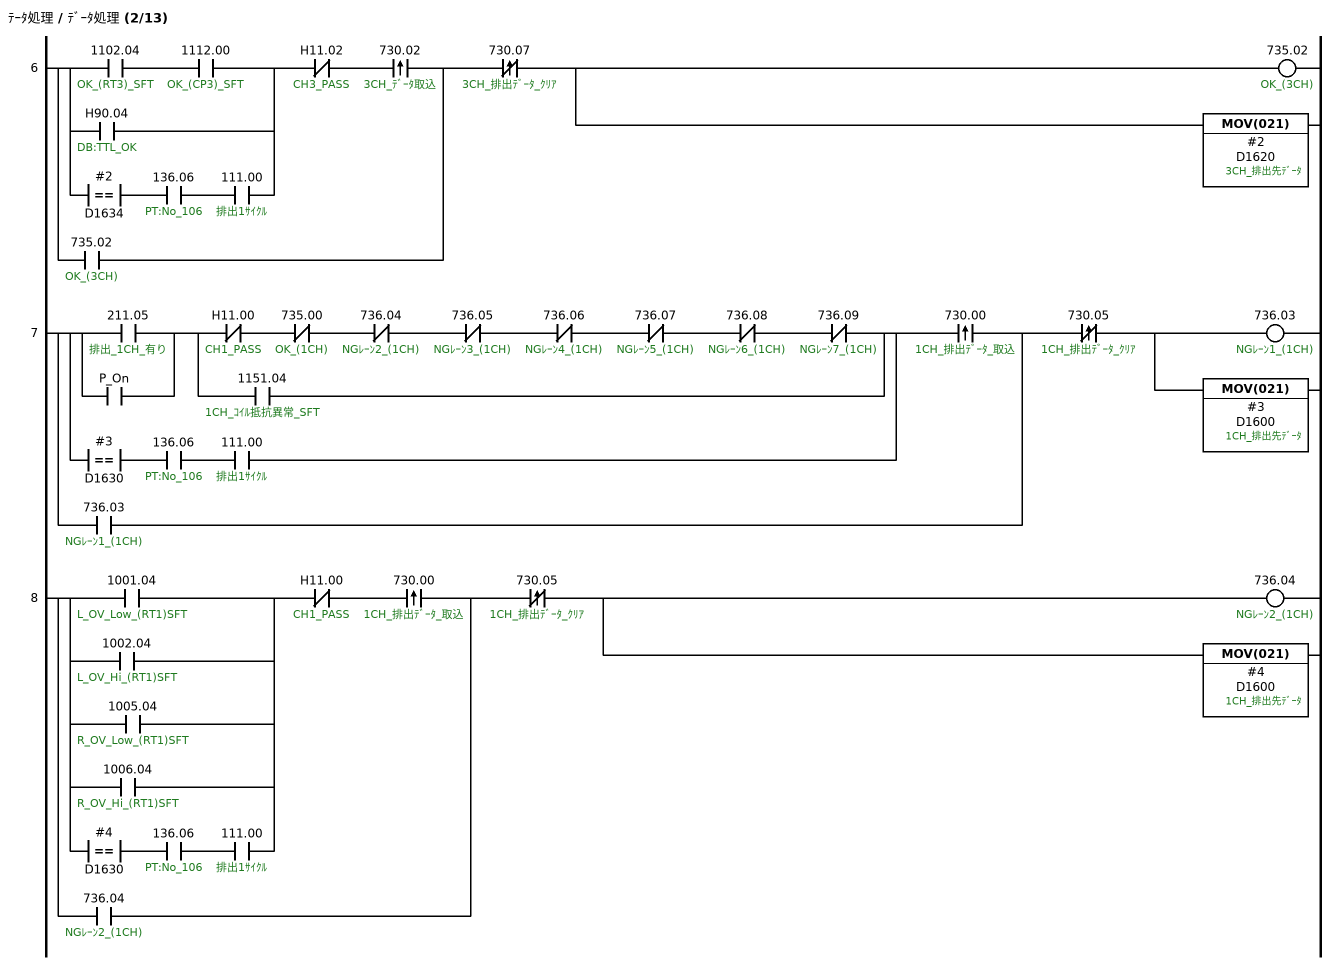
; rung 6
LD 1102.04  ; OK_(RT3)_SFT
AND 1112.00  ; OK_(CP3)_SFT
OR H90.04  ; DB:TTL_OK
LD=(300) #2 D1634
AND 136.06  ; PT:No_106
AND 111.00  ; 排出1ｻｲｸﾙ
ORLD
ANDNOT H11.02  ; CH3_PASS
@AND 730.02  ; 3CH_ﾃﾞｰﾀ取込
OR 735.02  ; OK_(3CH)
@ANDNOT 730.07  ; 3CH_排出ﾃﾞｰﾀ_ｸﾘｱ
OUT 735.02  ; OK_(3CH)
MOV(021) #2 D1620  ; 3CH_排出先ﾃﾞｰﾀ
; rung 7
LD 211.05  ; 排出_1CH_有り
OR P_On
LDNOT H11.00  ; CH1_PASS
ANDNOT 735.00  ; OK_(1CH)
ANDNOT 736.04  ; NGﾚｰﾝ2_(1CH)
ANDNOT 736.05  ; NGﾚｰﾝ3_(1CH)
ANDNOT 736.06  ; NGﾚｰﾝ4_(1CH)
ANDNOT 736.07  ; NGﾚｰﾝ5_(1CH)
ANDNOT 736.08  ; NGﾚｰﾝ6_(1CH)
ANDNOT 736.09  ; NGﾚｰﾝ7_(1CH)
OR 1151.04  ; 1CH_ｺｲﾙ抵抗異常_SFT
ANDLD
LD=(300) #3 D1630
AND 136.06  ; PT:No_106
AND 111.00  ; 排出1ｻｲｸﾙ
ORLD
@AND 730.00  ; 1CH_排出ﾃﾞｰﾀ_取込
OR 736.03  ; NGﾚｰﾝ1_(1CH)
@ANDNOT 730.05  ; 1CH_排出ﾃﾞｰﾀ_ｸﾘｱ
OUT 736.03  ; NGﾚｰﾝ1_(1CH)
MOV(021) #3 D1600  ; 1CH_排出先ﾃﾞｰﾀ
; rung 8
LD 1001.04  ; L_OV_Low_(RT1)SFT
OR 1002.04  ; L_OV_Hi_(RT1)SFT
OR 1005.04  ; R_OV_Low_(RT1)SFT
OR 1006.04  ; R_OV_Hi_(RT1)SFT
LD=(300) #4 D1630
AND 136.06  ; PT:No_106
AND 111.00  ; 排出1ｻｲｸﾙ
ORLD
ANDNOT H11.00  ; CH1_PASS
@AND 730.00  ; 1CH_排出ﾃﾞｰﾀ_取込
OR 736.04  ; NGﾚｰﾝ2_(1CH)
@ANDNOT 730.05  ; 1CH_排出ﾃﾞｰﾀ_ｸﾘｱ
OUT 736.04  ; NGﾚｰﾝ2_(1CH)
MOV(021) #4 D1600  ; 1CH_排出先ﾃﾞｰﾀ

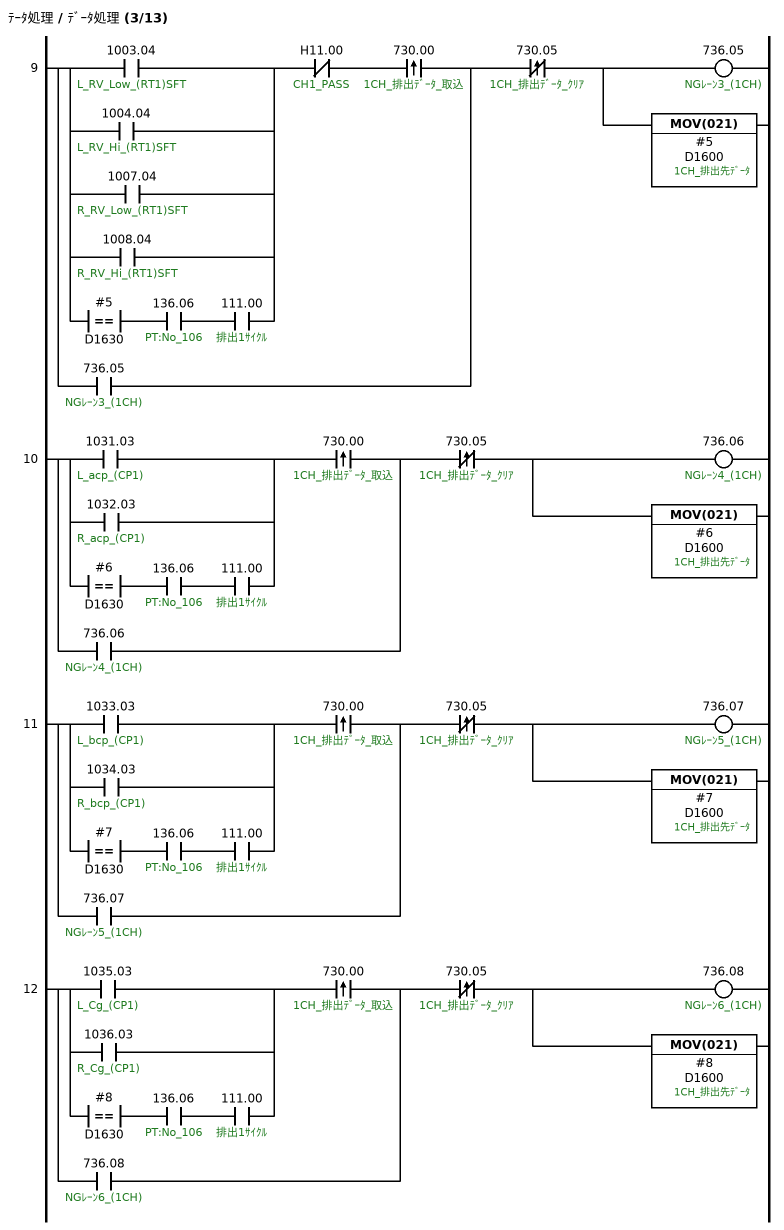
; rung 9
LD 1003.04  ; L_RV_Low_(RT1)SFT
OR 1004.04  ; L_RV_Hi_(RT1)SFT
OR 1007.04  ; R_RV_Low_(RT1)SFT
OR 1008.04  ; R_RV_Hi_(RT1)SFT
LD=(300) #5 D1630
AND 136.06  ; PT:No_106
AND 111.00  ; 排出1ｻｲｸﾙ
ORLD
ANDNOT H11.00  ; CH1_PASS
@AND 730.00  ; 1CH_排出ﾃﾞｰﾀ_取込
OR 736.05  ; NGﾚｰﾝ3_(1CH)
@ANDNOT 730.05  ; 1CH_排出ﾃﾞｰﾀ_ｸﾘｱ
OUT 736.05  ; NGﾚｰﾝ3_(1CH)
MOV(021) #5 D1600  ; 1CH_排出先ﾃﾞｰﾀ
; rung 10
LD 1031.03  ; L_acp_(CP1)
OR 1032.03  ; R_acp_(CP1)
LD=(300) #6 D1630
AND 136.06  ; PT:No_106
AND 111.00  ; 排出1ｻｲｸﾙ
ORLD
@AND 730.00  ; 1CH_排出ﾃﾞｰﾀ_取込
OR 736.06  ; NGﾚｰﾝ4_(1CH)
@ANDNOT 730.05  ; 1CH_排出ﾃﾞｰﾀ_ｸﾘｱ
OUT 736.06  ; NGﾚｰﾝ4_(1CH)
MOV(021) #6 D1600  ; 1CH_排出先ﾃﾞｰﾀ
; rung 11
LD 1033.03  ; L_bcp_(CP1)
OR 1034.03  ; R_bcp_(CP1)
LD=(300) #7 D1630
AND 136.06  ; PT:No_106
AND 111.00  ; 排出1ｻｲｸﾙ
ORLD
@AND 730.00  ; 1CH_排出ﾃﾞｰﾀ_取込
OR 736.07  ; NGﾚｰﾝ5_(1CH)
@ANDNOT 730.05  ; 1CH_排出ﾃﾞｰﾀ_ｸﾘｱ
OUT 736.07  ; NGﾚｰﾝ5_(1CH)
MOV(021) #7 D1600  ; 1CH_排出先ﾃﾞｰﾀ
; rung 12
LD 1035.03  ; L_Cg_(CP1)
OR 1036.03  ; R_Cg_(CP1)
LD=(300) #8 D1630
AND 136.06  ; PT:No_106
AND 111.00  ; 排出1ｻｲｸﾙ
ORLD
@AND 730.00  ; 1CH_排出ﾃﾞｰﾀ_取込
OR 736.08  ; NGﾚｰﾝ6_(1CH)
@ANDNOT 730.05  ; 1CH_排出ﾃﾞｰﾀ_ｸﾘｱ
OUT 736.08  ; NGﾚｰﾝ6_(1CH)
MOV(021) #8 D1600  ; 1CH_排出先ﾃﾞｰﾀ

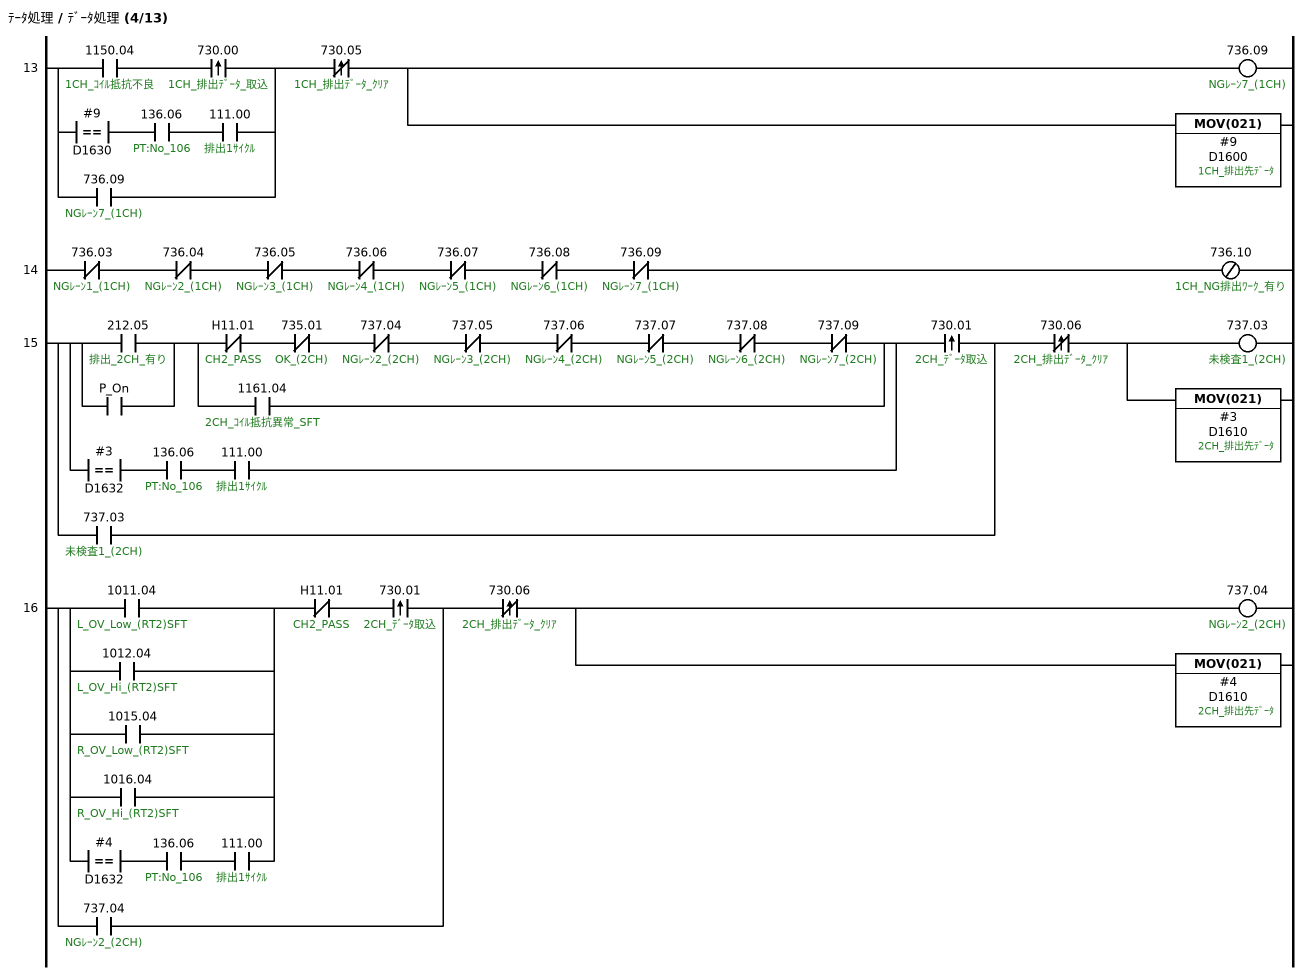
; rung 13
LD 1150.04  ; 1CH_ｺｲﾙ抵抗不良
@AND 730.00  ; 1CH_排出ﾃﾞｰﾀ_取込
LD=(300) #9 D1630
AND 136.06  ; PT:No_106
AND 111.00  ; 排出1ｻｲｸﾙ
ORLD
OR 736.09  ; NGﾚｰﾝ7_(1CH)
@ANDNOT 730.05  ; 1CH_排出ﾃﾞｰﾀ_ｸﾘｱ
OUT 736.09  ; NGﾚｰﾝ7_(1CH)
MOV(021) #9 D1600  ; 1CH_排出先ﾃﾞｰﾀ
; rung 14
LDNOT 736.03  ; NGﾚｰﾝ1_(1CH)
ANDNOT 736.04  ; NGﾚｰﾝ2_(1CH)
ANDNOT 736.05  ; NGﾚｰﾝ3_(1CH)
ANDNOT 736.06  ; NGﾚｰﾝ4_(1CH)
ANDNOT 736.07  ; NGﾚｰﾝ5_(1CH)
ANDNOT 736.08  ; NGﾚｰﾝ6_(1CH)
ANDNOT 736.09  ; NGﾚｰﾝ7_(1CH)
OUTNOT 736.10  ; 1CH_NG排出ﾜｰｸ_有り
; rung 15
LD 212.05  ; 排出_2CH_有り
OR P_On
LDNOT H11.01  ; CH2_PASS
ANDNOT 735.01  ; OK_(2CH)
ANDNOT 737.04  ; NGﾚｰﾝ2_(2CH)
ANDNOT 737.05  ; NGﾚｰﾝ3_(2CH)
ANDNOT 737.06  ; NGﾚｰﾝ4_(2CH)
ANDNOT 737.07  ; NGﾚｰﾝ5_(2CH)
ANDNOT 737.08  ; NGﾚｰﾝ6_(2CH)
ANDNOT 737.09  ; NGﾚｰﾝ7_(2CH)
OR 1161.04  ; 2CH_ｺｲﾙ抵抗異常_SFT
ANDLD
LD=(300) #3 D1632
AND 136.06  ; PT:No_106
AND 111.00  ; 排出1ｻｲｸﾙ
ORLD
@AND 730.01  ; 2CH_ﾃﾞｰﾀ取込
OR 737.03  ; 未検査1_(2CH)
@ANDNOT 730.06  ; 2CH_排出ﾃﾞｰﾀ_ｸﾘｱ
OUT 737.03  ; 未検査1_(2CH)
MOV(021) #3 D1610  ; 2CH_排出先ﾃﾞｰﾀ
; rung 16
LD 1011.04  ; L_OV_Low_(RT2)SFT
OR 1012.04  ; L_OV_Hi_(RT2)SFT
OR 1015.04  ; R_OV_Low_(RT2)SFT
OR 1016.04  ; R_OV_Hi_(RT2)SFT
LD=(300) #4 D1632
AND 136.06  ; PT:No_106
AND 111.00  ; 排出1ｻｲｸﾙ
ORLD
ANDNOT H11.01  ; CH2_PASS
@AND 730.01  ; 2CH_ﾃﾞｰﾀ取込
OR 737.04  ; NGﾚｰﾝ2_(2CH)
@ANDNOT 730.06  ; 2CH_排出ﾃﾞｰﾀ_ｸﾘｱ
OUT 737.04  ; NGﾚｰﾝ2_(2CH)
MOV(021) #4 D1610  ; 2CH_排出先ﾃﾞｰﾀ

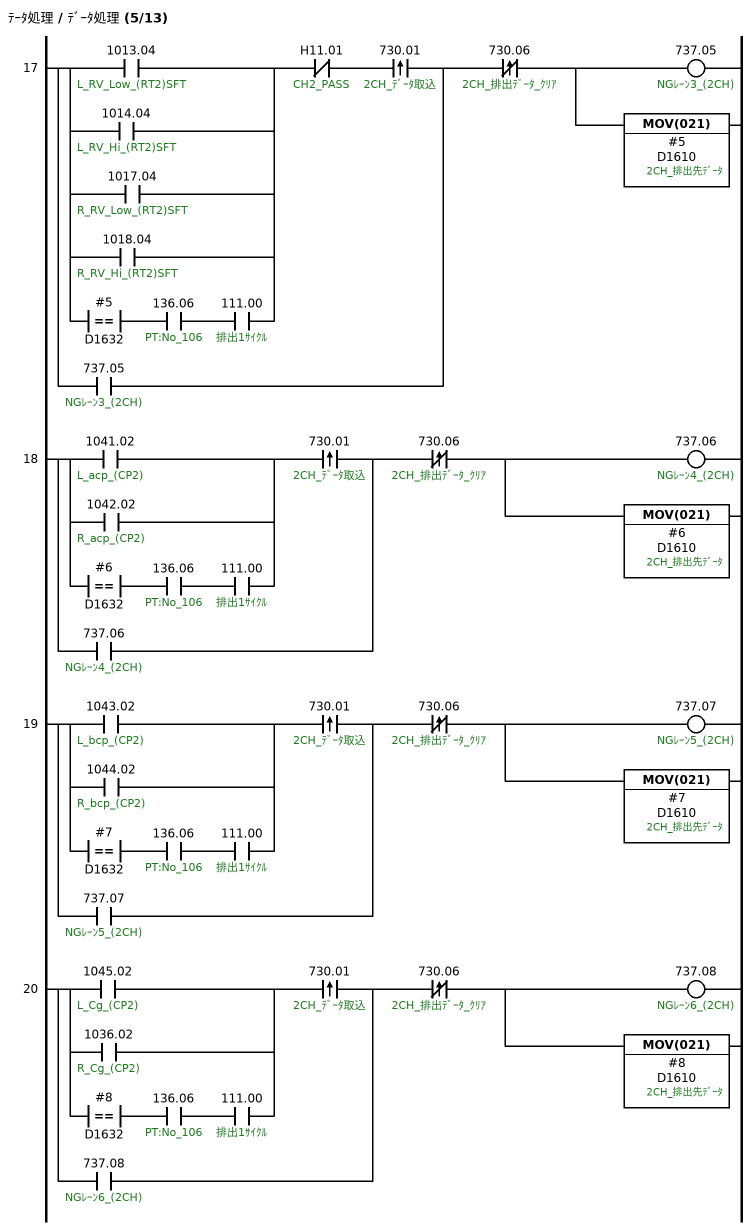
; rung 17
LD 1013.04  ; L_RV_Low_(RT2)SFT
OR 1014.04  ; L_RV_Hi_(RT2)SFT
OR 1017.04  ; R_RV_Low_(RT2)SFT
OR 1018.04  ; R_RV_Hi_(RT2)SFT
LD=(300) #5 D1632
AND 136.06  ; PT:No_106
AND 111.00  ; 排出1ｻｲｸﾙ
ORLD
ANDNOT H11.01  ; CH2_PASS
@AND 730.01  ; 2CH_ﾃﾞｰﾀ取込
OR 737.05  ; NGﾚｰﾝ3_(2CH)
@ANDNOT 730.06  ; 2CH_排出ﾃﾞｰﾀ_ｸﾘｱ
OUT 737.05  ; NGﾚｰﾝ3_(2CH)
MOV(021) #5 D1610  ; 2CH_排出先ﾃﾞｰﾀ
; rung 18
LD 1041.02  ; L_acp_(CP2)
OR 1042.02  ; R_acp_(CP2)
LD=(300) #6 D1632
AND 136.06  ; PT:No_106
AND 111.00  ; 排出1ｻｲｸﾙ
ORLD
@AND 730.01  ; 2CH_ﾃﾞｰﾀ取込
OR 737.06  ; NGﾚｰﾝ4_(2CH)
@ANDNOT 730.06  ; 2CH_排出ﾃﾞｰﾀ_ｸﾘｱ
OUT 737.06  ; NGﾚｰﾝ4_(2CH)
MOV(021) #6 D1610  ; 2CH_排出先ﾃﾞｰﾀ
; rung 19
LD 1043.02  ; L_bcp_(CP2)
OR 1044.02  ; R_bcp_(CP2)
LD=(300) #7 D1632
AND 136.06  ; PT:No_106
AND 111.00  ; 排出1ｻｲｸﾙ
ORLD
@AND 730.01  ; 2CH_ﾃﾞｰﾀ取込
OR 737.07  ; NGﾚｰﾝ5_(2CH)
@ANDNOT 730.06  ; 2CH_排出ﾃﾞｰﾀ_ｸﾘｱ
OUT 737.07  ; NGﾚｰﾝ5_(2CH)
MOV(021) #7 D1610  ; 2CH_排出先ﾃﾞｰﾀ
; rung 20
LD 1045.02  ; L_Cg_(CP2)
OR 1036.02  ; R_Cg_(CP2)
LD=(300) #8 D1632
AND 136.06  ; PT:No_106
AND 111.00  ; 排出1ｻｲｸﾙ
ORLD
@AND 730.01  ; 2CH_ﾃﾞｰﾀ取込
OR 737.08  ; NGﾚｰﾝ6_(2CH)
@ANDNOT 730.06  ; 2CH_排出ﾃﾞｰﾀ_ｸﾘｱ
OUT 737.08  ; NGﾚｰﾝ6_(2CH)
MOV(021) #8 D1610  ; 2CH_排出先ﾃﾞｰﾀ

